// TIA Portal project "Tia-portal-PLC" (V16)

(* hardware
DEVICE "S71500/ET200MP station_1"  S7-1500 station
   slot 0: "Rail_0"  Rack  6ES7 590-1***0-0AA0
   slot 1: "PLC_1"  CPU 1512C-1 PN  6ES7 512-1CK01-0AB0  V2.8
      slot 3: "CPU display_1"  6ES7591-1AA00-0AA0
      slot 32768: "PROFINET interface_1"  X1
         slot 32769: "Port_1"  X1 P1
         slot 32770: "Port_2"  X1 P2
      slot 34817: "Virtual CP interface port_1"  Virtual CP interface port  Virtual CP interface port
DEVICE "S71500/ET200MP station_2"  S7-1500 station
   slot 0: "Rail_0"  Rack  6ES7 590-1***0-0AA0
   slot 1: "PLC_2"  CPU 1512C-1 PN  6ES7 512-1CK01-0AB0  V2.8
      slot 3: "CPU display_1"  6ES7591-1AA00-0AA0
      slot 32768: "PROFINET interface_1"  X1
         slot 32769: "Port_1"  X1 P1
         slot 32770: "Port_2"  X1 P2
      slot 34817: "Virtual CP interface port_1"  Virtual CP interface port  Virtual CP interface port
DEVICE "HMI_1"  TP700 Comfort
   slot 0: "HMI_1"  TP700 Comfort  6AV2 124-0GC01-0AX0  16.0.0.0
   slot 1: "HMI_RT_1"  TP700 Comfort  6AV2 124-0GC01-0AX0  16.0.0.0
   slot 5: "HMI_1.IE_CP_1"  PROFINET Interface  16.0.0.0
      slot 1: "PROFINET Interface_1"  PROFINET Interface
         slot 1: "Port_1"  Port
         slot 2: "Port_2"  Port
   slot 7: "HMI_1.MPI/DP_CP_1"  MPI/DP Interface  16.0.0.0
*)

// ===== PLC "PLC_1"  CPU 1512C-1 PN =====

VAR_GLOBAL   // PLC tag table "Default tag table"
   "Tag_1" AT %M0.0 : Bool;
END_VAR

VAR_GLOBAL   // PLC tag table "Inputs"
   "Start_pos" AT %I0.0 : Bool;   // Item in starting position
   "Size_measure_pos" AT %I0.1 : Bool;   // Item in size measuring position
   "Weight_mes_pos" AT %I0.2 : Bool;   // Item in weight measuring pisition
   "Servo_table_pos" AT %I0.3 : Bool;   // Item on servo controlled table
   "Metal_sensor" AT %I0.4 : Bool;   // Inductive sensor
   "Grip_cyl_end_ext" AT %I0.5 : Bool;   // Reed sensor. Gripping cylinder in end position is extended
   "Grip_cyl_end_ret" AT %I0.6 : Bool;   // Reed sensor. Gripping cylinder in end position is retracted
   "Cyl_at_table_ext" AT %I0.7 : Bool;   // Reed sensor. Cylinder, pushing in bin is extended
   "Cyl_at_table_ret" AT %I1.0 : Bool;   // Reed sensor. Cylinder, pushing in bin is retracted
   "ES1" AT %I1.7 : Bool;   // Emergency stop button for measuring
   "ES2" AT %I2.0 : Bool;   // Emergency stop button for sorting
   "Size_measure" AT %IW0 : Int;   // Size measuring sensor
   "Load_cell" AT %IW2 : Int;   // Load cell
   "Grip_cyl_start_ext" AT %I2.1 : Bool;   // Reed sensor. Gripping cylinder in starting position is extended
   "Grip_cyl_start_ret" AT %I2.2 : Bool;   // Reed sensor. Gripping cylinder in starting position is retracted
   "Control24VButton" AT %I2.3 : Bool;   // Giving 24V supply for output moduls
   "Metal_measure_pos" AT %I2.4 : Bool;   // Item in metal measuring position
   "End_pos_at_conveyor" AT %I2.5 : Bool;   // Item in end position at inverter controlled conveyor
END_VAR

VAR_GLOBAL   // PLC tag table "Outputs"
   "Green_light" AT %Q4.0 : Bool;   // Green light
   "Yellow_light" AT %Q4.1 : Bool;   // Yellow light
   "Red_light" AT %Q4.2 : Bool;   // Red light
   "Move_grip_cyl_end_fwd" AT %Q4.3 : Bool;   // Extend gripping cylinder in end position
   "Move_grip_cyl_end_bwd" AT %Q4.4 : Bool;   // Retract gripping cylinder in end position
   "Move_cyl_at_table_fwd" AT %Q4.5 : Bool;   // Extend cylinder 1 for bin
   "Move_cyl_at_table_bwd" AT %Q4.6 : Bool;   // Retract cylinder 1 for bin
   "Conveyor_forward" AT %Q5.5 : Bool;   // Output for the inverter. Move conveyor forward
   "Conveyor_backward" AT %Q5.6 : Bool;   // Output for the inverter. Move conveyor backward
   "Move_grip_cyl_start_fwd" AT %Q5.7 : Bool;   // Extend gripping cylinder in start position
   "Move_grip_cyl_start_bwd" AT %Q6.0 : Bool;   // Retract gripping cylinder in start position
   "Blue_light" AT %Q4.7 : Bool;
END_VAR

DATA_BLOCK "HMI-data"   // DB2
{ S7_Optimized_Access := 'TRUE' }
VERSION : 0.1
   VAR
      AutomaticMode : Bool;
      StartConveyor : Bool;
      StopConveyor : Bool;
      ItemInTheSystem : Bool;   // If there is an item in the system
      TableAtHome : Bool;
      TableAtBin1 : Bool;
      TableAtBin2 : Bool;
      TableAtBin3 : Bool;
      TableAtBin4 : Bool;
      ES1NC : Bool := true;   // Emergency button for simulation
      ES2NC : Bool := true;   // Emergency button for simulation
      ControlSupplyOK : Bool;   // Control 24V for simulation
      SizeInCm : Real;
      MetalMaterial : Bool;
      WeightInKg : Real;
      Bin1Breed : Bool;   // Small and non metal
      Bin2Breed : Bool;   // Small and metal
      Bin3Breed : Bool;   // Large and not metal
      Bin4Breed : Bool;   // Large and metal
      HomePosition : LReal;
      Bin1Position : LReal := 30.0;
      Bin2Position : LReal := 60.0;
      Bin3Postion : LReal := 90.0;
      Bin4Position : LReal := 120.0;
   END_VAR
BEGIN
END_DATA_BLOCK

DATA_BLOCK "OPCUA-data"   // DB4
{ S7_Optimized_Access := 'FALSE' }
VERSION : 0.1
   VAR
      Sensor1 : Bool := true;
   END_VAR
BEGIN
END_DATA_BLOCK

DATA_BLOCK "Sorting-motion-control_DB"   // DB7
{ S7_Optimized_Access := 'TRUE' }
VERSION : 0.1
// stored: InstanceOfName Sorting-motion-control
"Sorting-motion-control"
BEGIN
END_DATA_BLOCK

DATA_BLOCK "Size-measure_DB"   // DB8
{ S7_Optimized_Access := 'TRUE' }
VERSION : 0.1
// stored: InstanceOfName Size-measure
"Size-measure"
BEGIN
END_DATA_BLOCK

DATA_BLOCK "Weight-measure_DB"   // DB9
{ S7_Optimized_Access := 'TRUE' }
VERSION : 0.1
// stored: InstanceOfName Weight-measure
"Weight-measure"
BEGIN
END_DATA_BLOCK

DATA_BLOCK "Bin-sensors-from-PLC2"   // DB14
{ S7_Optimized_Access := 'FALSE' }
VERSION : 0.1
   VAR
      Bin1Full : Bool;
      Bin2Full : Bool;
      Bin3Full : Bool;
      Bin4Full : Bool;
   END_VAR
BEGIN
END_DATA_BLOCK

DATA_BLOCK "PLC2-communication_DB"   // DB16
{ S7_Optimized_Access := 'TRUE' }
VERSION : 0.1
// stored: InstanceOfName PLC2-communication
"PLC2-communication"
BEGIN
END_DATA_BLOCK

// folder: System blocks/Program resources

DATA_BLOCK "Start-pos-timer-DB"   // DB3
{ S7_Optimized_Access := 'TRUE' }
AUTHOR : Simatic
FAMILY : IEC
NAME : IEC_TMR
VERSION : 1.0
// stored: InstanceOfName IEC_TIMER
"IEC_TIMER"
BEGIN
END_DATA_BLOCK

DATA_BLOCK "IEC_Timer_0_DB"   // DB5
{ S7_Optimized_Access := 'TRUE' }
AUTHOR : Simatic
FAMILY : IEC
NAME : IEC_TMR
VERSION : 1.0
// stored: InstanceOfName IEC_TIMER
"IEC_TIMER"
BEGIN
END_DATA_BLOCK

DATA_BLOCK "IEC_Timer_0_DB_1"   // DB6
{ S7_Optimized_Access := 'TRUE' }
AUTHOR : Simatic
FAMILY : IEC
NAME : IEC_TMR
VERSION : 1.0
// stored: InstanceOfName IEC_TIMER
"IEC_TIMER"
BEGIN
END_DATA_BLOCK

DATA_BLOCK "IEC_Timer_0_DB_2"   // DB10
{ S7_Optimized_Access := 'TRUE' }
AUTHOR : Simatic
FAMILY : IEC
NAME : IEC_TMR
VERSION : 1.0
// stored: InstanceOfName IEC_TIMER
"IEC_TIMER"
BEGIN
END_DATA_BLOCK

DATA_BLOCK "IEC_Timer_0_DB_3"   // DB11
{ S7_Optimized_Access := 'TRUE' }
AUTHOR : Simatic
FAMILY : IEC
NAME : IEC_TMR
VERSION : 1.0
// stored: InstanceOfName IEC_TIMER
"IEC_TIMER"
BEGIN
END_DATA_BLOCK

DATA_BLOCK "IEC_Timer_0_DB_5"   // DB13
{ S7_Optimized_Access := 'TRUE' }
AUTHOR : Simatic
FAMILY : IEC
NAME : IEC_TMR
VERSION : 1.0
// stored: InstanceOfName IEC_TIMER
"IEC_TIMER"
BEGIN
END_DATA_BLOCK

DATA_BLOCK "PLC_1_Receive_DB"   // DB15
{ S7_Optimized_Access := 'TRUE' }
AUTHOR : SIMATIC
FAMILY : MC7Plus
NAME : TC_IP_v4
VERSION : 1.0
// stored: InstanceOfName TCON_IP_v4
"TCON_IP_v4"
BEGIN
   ID := 1;
   InterfaceId := 64;
   LocalPort := 2000;
   RemoteAddress.ADDR[1] := 192;
   RemoteAddress.ADDR[2] := 168;
   RemoteAddress.ADDR[4] := 14;
END_DATA_BLOCK

DATA_BLOCK "IEC_Timer_0_DB_8"   // DB17
{ S7_Optimized_Access := 'TRUE' }
AUTHOR : Simatic
FAMILY : IEC
NAME : IEC_TMR
VERSION : 1.0
// stored: InstanceOfName IEC_TIMER
"IEC_TIMER"
BEGIN
END_DATA_BLOCK

DATA_BLOCK "IEC_Timer_0_DB_6"   // DB18
{ S7_Optimized_Access := 'TRUE' }
AUTHOR : Simatic
FAMILY : IEC
NAME : IEC_TMR
VERSION : 1.0
// stored: InstanceOfName IEC_TIMER
"IEC_TIMER"
BEGIN
END_DATA_BLOCK

DATA_BLOCK "IEC_Timer_0_DB_7"   // DB19
{ S7_Optimized_Access := 'TRUE' }
AUTHOR : Simatic
FAMILY : IEC
NAME : IEC_TMR
VERSION : 1.0
// stored: InstanceOfName IEC_TIMER
"IEC_TIMER"
BEGIN
END_DATA_BLOCK

// folder: (top level)

DATA_BLOCK "SortingAxis_1"   // DB1, Motion_DB
{ S7_Optimized_Access := 'TRUE' }
AUTHOR : SIMATIC
FAMILY : MC_1500
VERSION : 5.0
// stored: InstanceOfName TO_PositioningAxis
"TO_PositioningAxis"
BEGIN
END_DATA_BLOCK

FUNCTION_BLOCK "Sorting-motion-control"   // FB1, LAD
{ S7_Optimized_Access := 'TRUE' }
VERSION : 0.1
   VAR_INPUT
      EnablePower : Bool;
      ExecuteReset : Bool;
      ExecuteHome : Bool;
      ExecuteHalt : Bool;
      JogFwd : Bool;
      JogBwd : Bool;
      JogVelocity : LReal;
      ExecuteMoveVelocity : Bool;
      McVelocity : LReal;
      ExecuteMoveRelative : Bool;
      MoveRelativeValue : LReal;
      ExecuteMoveAbsolute : Bool;
      MoveAbsoluteValue : LReal;
      ExecuteStop : Bool;
   END_VAR
   VAR_OUTPUT
      ActualPosition : LReal;
      ActualSpeed : LReal;
      ActualVelocity : LReal;
   END_VAR
   VAR
      MC_POWER_Instance : MC_POWER;
      MC_RESET_Instance : MC_RESET;
      MC_HOME_Instance : MC_HOME;
      MC_HALT_Instance : MC_HALT;
      MC_MOVEJOG_Instance : MC_MOVEJOG;
      MC_MOVEVELOCITY_Instance : MC_MOVEVELOCITY;
      MC_MOVERELATIVE_Instance : MC_MOVERELATIVE;
      MC_MOVEABSOLUTE_Instance : MC_MOVEABSOLUTE;
      MC_STOP_Instance : MC_STOP;
   END_VAR
BEGIN

REGION Network 1: MC Power
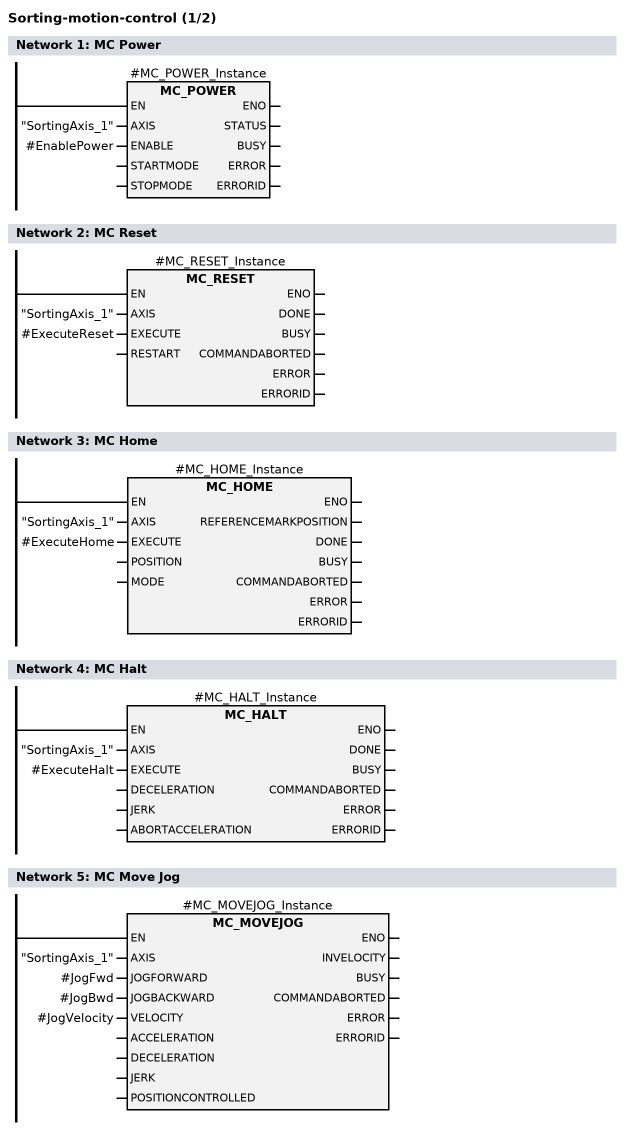
   #MC_POWER_Instance(Axis := "SortingAxis_1", Enable := #EnablePower);   // MC_POWER
END_REGION

REGION Network 2: MC Reset
   #MC_RESET_Instance(Axis := "SortingAxis_1", Execute := #ExecuteReset);   // MC_RESET
END_REGION

REGION Network 3: MC Home
   #MC_HOME_Instance(Axis := "SortingAxis_1", Execute := #ExecuteHome);   // MC_HOME
END_REGION

REGION Network 4: MC Halt
   #MC_HALT_Instance(Axis := "SortingAxis_1", Execute := #ExecuteHalt);   // MC_HALT
END_REGION

REGION Network 5: MC Move Jog
   #MC_MOVEJOG_Instance(Axis := "SortingAxis_1",   // MC_MOVEJOG
                        JogForward := #JogFwd,
                        JogBackward := #JogBwd,
                        Velocity := #JogVelocity);
END_REGION

REGION Network 6: MC Move Velocity
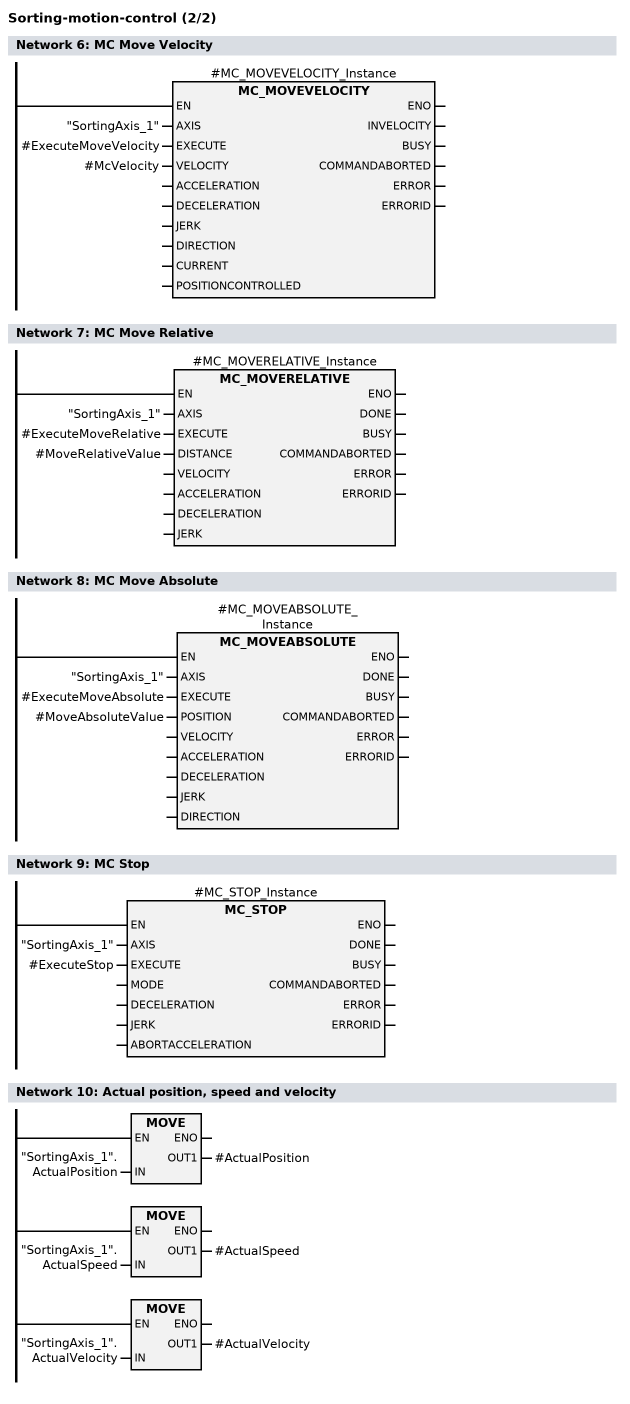
   #MC_MOVEVELOCITY_Instance(Axis := "SortingAxis_1", Execute := #ExecuteMoveVelocity, Velocity := #McVelocity);   // MC_MOVEVELOCITY
END_REGION

REGION Network 7: MC Move Relative
   #MC_MOVERELATIVE_Instance(Axis := "SortingAxis_1",   // MC_MOVERELATIVE
                           Execute := #ExecuteMoveRelative,
                           Distance := #MoveRelativeValue);
END_REGION

REGION Network 8: MC Move Absolute
   #MC_MOVEABSOLUTE_Instance(Axis := "SortingAxis_1",   // MC_MOVEABSOLUTE
                           Execute := #ExecuteMoveAbsolute,
                           Position := #MoveAbsoluteValue);
END_REGION

REGION Network 9: MC Stop
   #MC_STOP_Instance(Axis := "SortingAxis_1", Execute := #ExecuteStop);   // MC_STOP
END_REGION

REGION Network 10: Actual position, speed and velocity
   RUNG wire#powerrail
      Move(in := "SortingAxis_1".ActualPosition, out1 => #ActualPosition)
   END_RUNG
   RUNG wire#powerrail
      Move(in := "SortingAxis_1".ActualSpeed, out1 => #ActualSpeed)
   END_RUNG
   RUNG wire#powerrail
      Move(in := "SortingAxis_1".ActualVelocity, out1 => #ActualVelocity)
   END_RUNG
   // the same network as SCL:
   #ActualPosition := "SortingAxis_1".ActualPosition;
   #ActualSpeed := "SortingAxis_1".ActualSpeed;
   #ActualVelocity := "SortingAxis_1".ActualVelocity;
END_REGION
END_FUNCTION_BLOCK

FUNCTION_BLOCK "Size-measure"   // FB2, LAD
{ S7_Optimized_Access := 'TRUE' }
VERSION : 0.1
   VAR_INPUT
      TestValue : Int := 0;
   END_VAR
   VAR_OUTPUT
      SizeInCm : Real;
   END_VAR
   VAR_TEMP
      SizeInPercent : Real;
   END_VAR
BEGIN

REGION Network 1
   // Converting analog voltage to percent
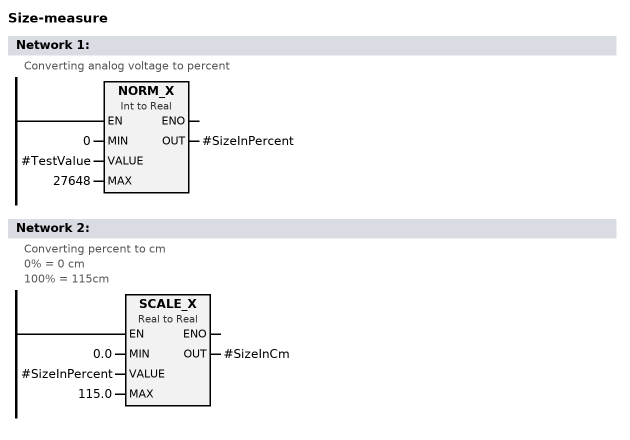
   RUNG wire#powerrail
      { S7_Templates := "[SrcType := Int, DestType := Real]" } Normalize(min := 0, value := #TestValue, max := 27648, out => #SizeInPercent)
   END_RUNG
   // the same network as SCL:
   #SizeInPercent := NORM_X(MIN := 0, VALUE := #TestValue, MAX := 27648);
END_REGION

REGION Network 2
   // Converting percent to cm
   // 0% = 0 cm
   // 100% = 115cm
   RUNG wire#powerrail
      { S7_Templates := "[SrcType := Real, DestType := Real]" } Scale(min := 0.0, value := #SizeInPercent, max := 115.0, out => #SizeInCm)
   END_RUNG
   // the same network as SCL:
   #SizeInCm := SCALE_X(MIN := 0.0, VALUE := #SizeInPercent, MAX := 115.0);
END_REGION
END_FUNCTION_BLOCK

FUNCTION_BLOCK "Weight-measure"   // FB3, LAD
{ S7_Optimized_Access := 'TRUE' }
VERSION : 0.1
   VAR_INPUT
      TestValue : Int := 0;
   END_VAR
   VAR_OUTPUT
      WeightInKg : Real;
   END_VAR
   VAR_TEMP
      WeightInPercent : Real;
   END_VAR
BEGIN

REGION Network 1
   // Converting analog voltage to percent
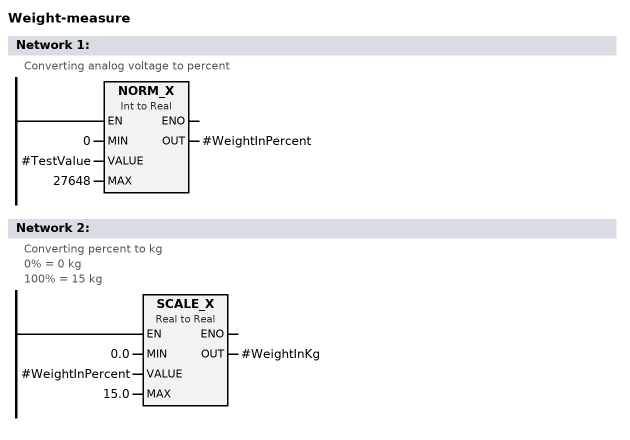
   RUNG wire#powerrail
      { S7_Templates := "[SrcType := Int, DestType := Real]" } Normalize(min := 0, value := #TestValue, max := 27648, out => #WeightInPercent)
   END_RUNG
   // the same network as SCL:
   #WeightInPercent := NORM_X(MIN := 0, VALUE := #TestValue, MAX := 27648);
END_REGION

REGION Network 2
   // Converting percent to kg
   // 0% = 0 kg
   // 100% = 15 kg
   RUNG wire#powerrail
      { S7_Templates := "[SrcType := Real, DestType := Real]" } Scale(min := 0.0, value := #WeightInPercent, max := 15.0, out => #WeightInKg)
   END_RUNG
   // the same network as SCL:
   #WeightInKg := SCALE_X(MIN := 0.0, VALUE := #WeightInPercent, MAX := 15.0);
END_REGION
END_FUNCTION_BLOCK

FUNCTION_BLOCK "PLC2-communication"   // FB4, LAD
TITLE = Communication with PLC2
{ S7_Optimized_Access := 'TRUE' }
VERSION : 0.1
   VAR_INPUT
      EnableConnAndRead : Bool;
   END_VAR
   VAR
      TRCV_C_Instance : TRCV_C;
   END_VAR
BEGIN

REGION Network 1
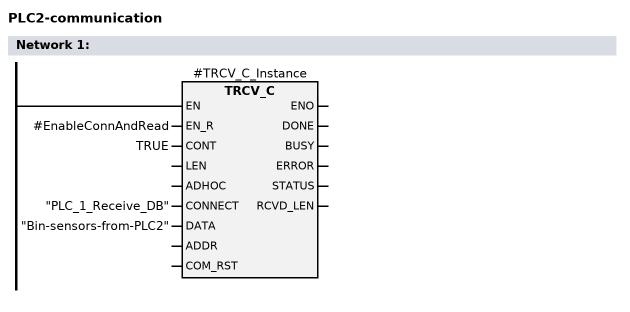
   #TRCV_C_Instance(EN_R := #EnableConnAndRead,   // TRCV_C
                    CONT := TRUE,
                    CONNECT := "PLC_1_Receive_DB",
                    DATA := "Bin-sensors-from-PLC2");
END_REGION
END_FUNCTION_BLOCK

FUNCTION "Home-positions" : Void   // FC1, LAD
{ S7_Optimized_Access := 'TRUE' }
VERSION : 0.1
// If there is 24V control power supply, everything goes to home position.
// If the ControlSupplyOK variable is true.
BEGIN

REGION Network 1: Extend gripping cylinder in start position
   // Gripping cylinder in start position is extended
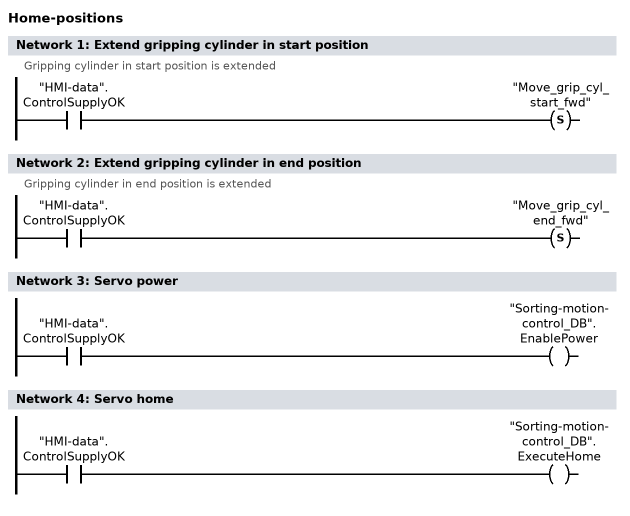
   RUNG wire#powerrail
      Contact( "HMI-data".ControlSupplyOK )
      S_Coil( "Move_grip_cyl_start_fwd" )
   END_RUNG
   // the same network as SCL:
   IF "HMI-data".ControlSupplyOK THEN "Move_grip_cyl_start_fwd" := TRUE; END_IF;
END_REGION

REGION Network 2: Extend gripping cylinder in end position
   // Gripping cylinder in end position is extended
   RUNG wire#powerrail
      Contact( "HMI-data".ControlSupplyOK )
      S_Coil( "Move_grip_cyl_end_fwd" )
   END_RUNG
   // the same network as SCL:
   IF "HMI-data".ControlSupplyOK THEN "Move_grip_cyl_end_fwd" := TRUE; END_IF;
END_REGION

REGION Network 3: Servo power
   RUNG wire#powerrail
      Contact( "HMI-data".ControlSupplyOK )
      Coil( "Sorting-motion-control_DB".EnablePower )
   END_RUNG
   // the same network as SCL:
   "Sorting-motion-control_DB".EnablePower := "HMI-data".ControlSupplyOK;
END_REGION

REGION Network 4: Servo home
   RUNG wire#powerrail
      Contact( "HMI-data".ControlSupplyOK )
      Coil( "Sorting-motion-control_DB".ExecuteHome )
   END_RUNG
   // the same network as SCL:
   "Sorting-motion-control_DB".ExecuteHome := "HMI-data".ControlSupplyOK;
END_REGION
END_FUNCTION

FUNCTION "Control24V" : Void   // FC2, LAD
{ S7_Optimized_Access := 'TRUE' }
VERSION : 0.1
BEGIN

REGION Network 1: Control 24V for simulation
   // This is the simulation of the safety circuit. Power supply for the output modules.
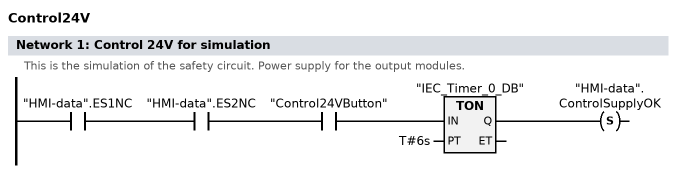
   "IEC_Timer_0_DB".TON(IN := "HMI-data".ES1NC AND "HMI-data".ES2NC AND "Control24VButton", PT := T#6s);
   IF "IEC_Timer_0_DB".Q THEN "HMI-data".ControlSupplyOK := TRUE; END_IF;
END_REGION
END_FUNCTION

FUNCTION "Table-positions" : Void   // FC3, LAD
{ S7_Optimized_Access := 'TRUE' }
VERSION : 0.1
BEGIN

REGION Network 1: Home position
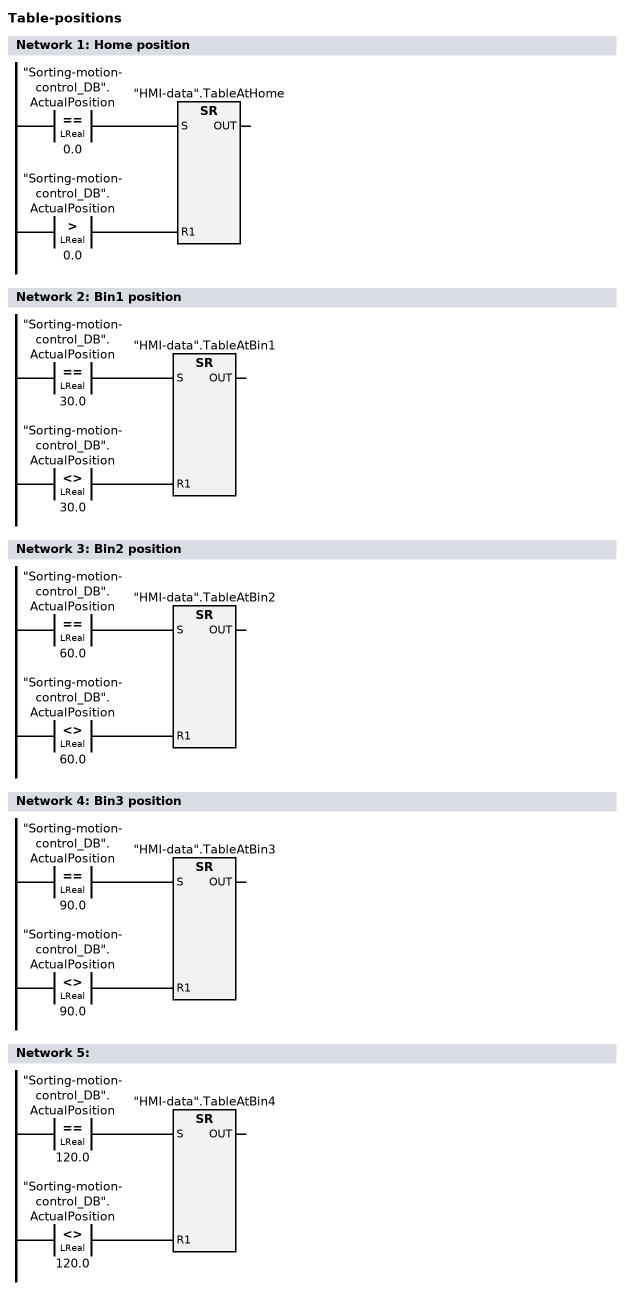
   RUNG wire#powerrail
      { S7_Templates := "SrcType := LReal" } EQ_Contact(in1 := "Sorting-motion-control_DB".ActualPosition, in2 := 0.0)
      S_SR(operand := "HMI-data".TableAtHome, r1 := wire#w1)
   END_RUNG
   RUNG wire#powerrail
      { S7_Templates := "SrcType := LReal" } GT_Contact(in1 := "Sorting-motion-control_DB".ActualPosition, in2 := 0.0)
   END_RUNG wire#w1
   // the same network as SCL:
   IF "Sorting-motion-control_DB".ActualPosition = 0.0 THEN
       "HMI-data".TableAtHome := TRUE;   // SR flip-flop
   END_IF;
   IF "Sorting-motion-control_DB".ActualPosition > 0.0 THEN "HMI-data".TableAtHome := FALSE; END_IF;
END_REGION

REGION Network 2: Bin1 position
   RUNG wire#powerrail
      { S7_Templates := "SrcType := LReal" } EQ_Contact(in1 := "Sorting-motion-control_DB".ActualPosition, in2 := 30.0)
      S_SR(operand := "HMI-data".TableAtBin1, r1 := wire#w1)
   END_RUNG
   RUNG wire#powerrail
      { S7_Templates := "SrcType := LReal" } NE_Contact(in1 := "Sorting-motion-control_DB".ActualPosition, in2 := 30.0)
   END_RUNG wire#w1
   // the same network as SCL:
   IF "Sorting-motion-control_DB".ActualPosition = 30.0 THEN
       "HMI-data".TableAtBin1 := TRUE;   // SR flip-flop
   END_IF;
   IF "Sorting-motion-control_DB".ActualPosition <> 30.0 THEN "HMI-data".TableAtBin1 := FALSE; END_IF;
END_REGION

REGION Network 3: Bin2 position
   RUNG wire#powerrail
      { S7_Templates := "SrcType := LReal" } EQ_Contact(in1 := "Sorting-motion-control_DB".ActualPosition, in2 := 60.0)
      S_SR(operand := "HMI-data".TableAtBin2, r1 := wire#w1)
   END_RUNG
   RUNG wire#powerrail
      { S7_Templates := "SrcType := LReal" } NE_Contact(in1 := "Sorting-motion-control_DB".ActualPosition, in2 := 60.0)
   END_RUNG wire#w1
   // the same network as SCL:
   IF "Sorting-motion-control_DB".ActualPosition = 60.0 THEN
       "HMI-data".TableAtBin2 := TRUE;   // SR flip-flop
   END_IF;
   IF "Sorting-motion-control_DB".ActualPosition <> 60.0 THEN "HMI-data".TableAtBin2 := FALSE; END_IF;
END_REGION

REGION Network 4: Bin3 position
   RUNG wire#powerrail
      { S7_Templates := "SrcType := LReal" } EQ_Contact(in1 := "Sorting-motion-control_DB".ActualPosition, in2 := 90.0)
      S_SR(operand := "HMI-data".TableAtBin3, r1 := wire#w1)
   END_RUNG
   RUNG wire#powerrail
      { S7_Templates := "SrcType := LReal" } NE_Contact(in1 := "Sorting-motion-control_DB".ActualPosition, in2 := 90.0)
   END_RUNG wire#w1
   // the same network as SCL:
   IF "Sorting-motion-control_DB".ActualPosition = 90.0 THEN
       "HMI-data".TableAtBin3 := TRUE;   // SR flip-flop
   END_IF;
   IF "Sorting-motion-control_DB".ActualPosition <> 90.0 THEN "HMI-data".TableAtBin3 := FALSE; END_IF;
END_REGION

REGION Network 5
   RUNG wire#powerrail
      { S7_Templates := "SrcType := LReal" } EQ_Contact(in1 := "Sorting-motion-control_DB".ActualPosition, in2 := 120.0)
      S_SR(operand := "HMI-data".TableAtBin4, r1 := wire#w1)
   END_RUNG
   RUNG wire#powerrail
      { S7_Templates := "SrcType := LReal" } NE_Contact(in1 := "Sorting-motion-control_DB".ActualPosition, in2 := 120.0)
   END_RUNG wire#w1
   // the same network as SCL:
   IF "Sorting-motion-control_DB".ActualPosition = 120.0 THEN
       "HMI-data".TableAtBin4 := TRUE;   // SR flip-flop
   END_IF;
   IF "Sorting-motion-control_DB".ActualPosition <> 120.0 THEN "HMI-data".TableAtBin4 := FALSE; END_IF;
END_REGION
END_FUNCTION

FUNCTION "Breed-calculation" : Void   // FC4, LAD
{ S7_Optimized_Access := 'TRUE' }
VERSION : 0.1
BEGIN

REGION Network 1: Small and non metal
   // Bin1 breed
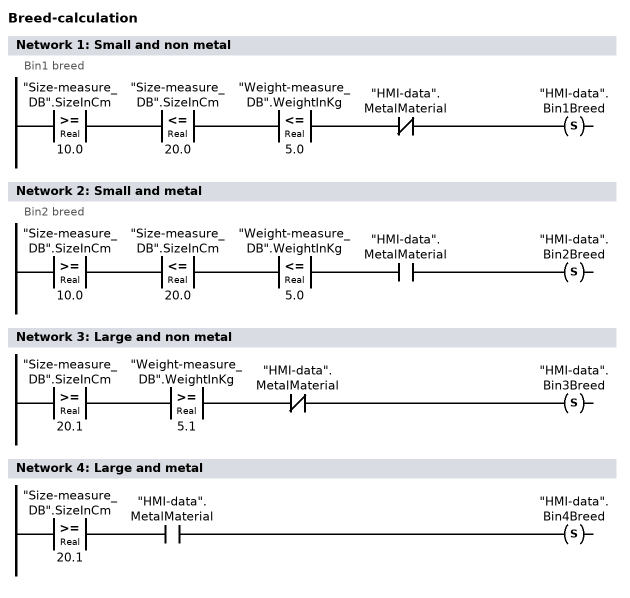
   RUNG wire#powerrail
      { S7_Templates := "SrcType := Real" } GE_Contact(in1 := "Size-measure_DB".SizeInCm, in2 := 10.0)
      { S7_Templates := "SrcType := Real" } LE_Contact(in1 := "Size-measure_DB".SizeInCm, in2 := 20.0)
      { S7_Templates := "SrcType := Real" } LE_Contact(in1 := "Weight-measure_DB".WeightInKg, in2 := 5.0)
      I_Contact( "HMI-data".MetalMaterial )
      S_Coil( "HMI-data".Bin1Breed )
   END_RUNG
   // the same network as SCL:
   IF ("Size-measure_DB".SizeInCm >= 10.0) AND ("Size-measure_DB".SizeInCm <= 20.0) AND ("Weight-measure_DB".WeightInKg <= 5.0) AND NOT "HMI-data".MetalMaterial THEN
       "HMI-data".Bin1Breed := TRUE;
   END_IF;
END_REGION

REGION Network 2: Small and metal
   // Bin2 breed
   RUNG wire#powerrail
      { S7_Templates := "SrcType := Real" } GE_Contact(in1 := "Size-measure_DB".SizeInCm, in2 := 10.0)
      { S7_Templates := "SrcType := Real" } LE_Contact(in1 := "Size-measure_DB".SizeInCm, in2 := 20.0)
      { S7_Templates := "SrcType := Real" } LE_Contact(in1 := "Weight-measure_DB".WeightInKg, in2 := 5.0)
      Contact( "HMI-data".MetalMaterial )
      S_Coil( "HMI-data".Bin2Breed )
   END_RUNG
   // the same network as SCL:
   IF ("Size-measure_DB".SizeInCm >= 10.0) AND ("Size-measure_DB".SizeInCm <= 20.0) AND ("Weight-measure_DB".WeightInKg <= 5.0) AND "HMI-data".MetalMaterial THEN
       "HMI-data".Bin2Breed := TRUE;
   END_IF;
END_REGION

REGION Network 3: Large and non metal
   RUNG wire#powerrail
      { S7_Templates := "SrcType := Real" } GE_Contact(in1 := "Size-measure_DB".SizeInCm, in2 := 20.1)
      { S7_Templates := "SrcType := Real" } GE_Contact(in1 := "Weight-measure_DB".WeightInKg, in2 := 5.1)
      I_Contact( "HMI-data".MetalMaterial )
      S_Coil( "HMI-data".Bin3Breed )
   END_RUNG
   // the same network as SCL:
   IF ("Size-measure_DB".SizeInCm >= 20.1) AND ("Weight-measure_DB".WeightInKg >= 5.1) AND NOT "HMI-data".MetalMaterial THEN
       "HMI-data".Bin3Breed := TRUE;
   END_IF;
END_REGION

REGION Network 4: Large and metal
   RUNG wire#powerrail
      { S7_Templates := "SrcType := Real" } GE_Contact(in1 := "Size-measure_DB".SizeInCm, in2 := 20.1)
      Contact( "HMI-data".MetalMaterial )
      S_Coil( "HMI-data".Bin4Breed )
   END_RUNG
   // the same network as SCL:
   IF ("Size-measure_DB".SizeInCm >= 20.1) AND "HMI-data".MetalMaterial THEN
       "HMI-data".Bin4Breed := TRUE;
   END_IF;
END_REGION
END_FUNCTION

ORGANIZATION_BLOCK "Main"   // OB1, LAD, ProgramCycle
TITLE = "Main Program Sweep (Cycle)"
{ S7_Optimized_Access := 'TRUE' }
VERSION : 0.1
   VAR_INPUT
      Initial_Call : Bool;   // Initial call of this OB
      Remanence : Bool;   // =True, if remanent data are available
   END_VAR
   VAR_TEMP   // added for the SCL form of the ladder/FBD networks
      _w1 : Bool;
      _w2 : Bool;
      _w3 : Bool;
      _w4 : Bool;
   END_VAR
BEGIN

REGION Network 1: Control 24V power supply
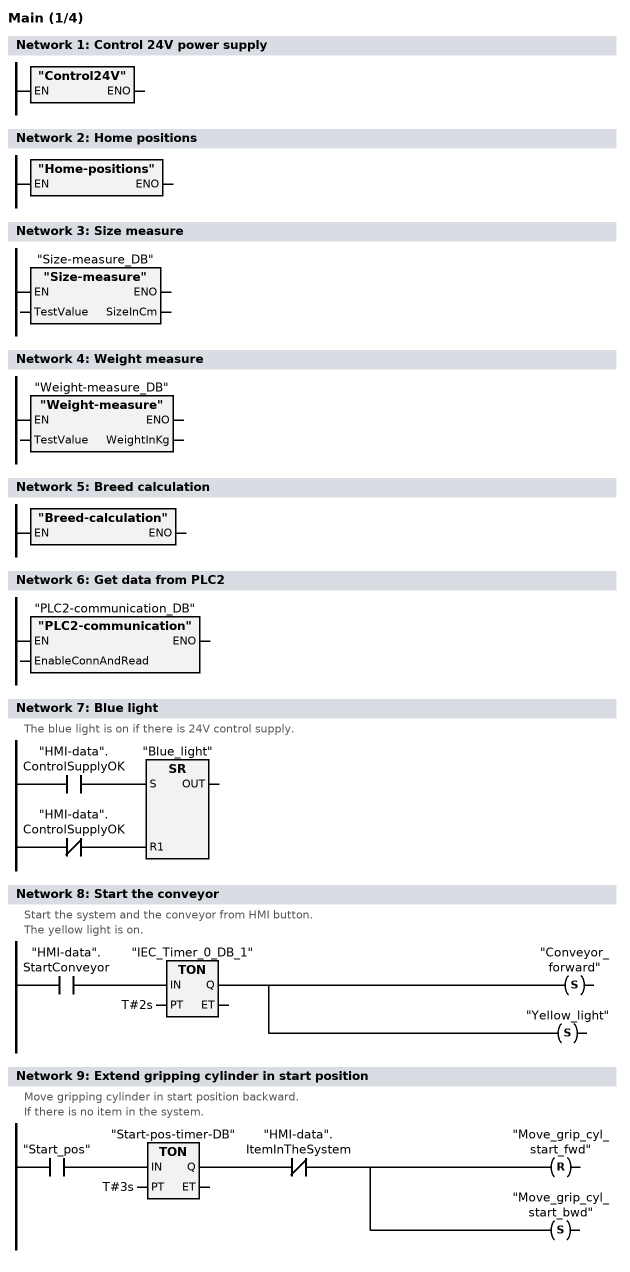
   RUNG wire#powerrail
      "Control24V"()
   END_RUNG
   // the same network as SCL:
   "Control24V"();
END_REGION

REGION Network 2: Home positions
   RUNG wire#powerrail
      "Home-positions"()
   END_RUNG
   // the same network as SCL:
   "Home-positions"();
END_REGION

REGION Network 3: Size measure
   RUNG wire#powerrail
      "Size-measure_DB"(TestValue :=, SizeInCm =>)
   END_RUNG
   // the same network as SCL:
   "Size-measure_DB"();   // "Size-measure"
END_REGION

REGION Network 4: Weight measure
   RUNG wire#powerrail
      "Weight-measure_DB"(TestValue :=, WeightInKg =>)
   END_RUNG
   // the same network as SCL:
   "Weight-measure_DB"();   // "Weight-measure"
END_REGION

REGION Network 5: Breed calculation
   RUNG wire#powerrail
      "Breed-calculation"()
   END_RUNG
   // the same network as SCL:
   "Breed-calculation"();
END_REGION

REGION Network 6: Get data from PLC2
   RUNG wire#powerrail
      "PLC2-communication_DB"(EnableConnAndRead :=)
   END_RUNG
   // the same network as SCL:
   "PLC2-communication_DB"();   // "PLC2-communication"
END_REGION

REGION Network 7: Blue light
   // The blue light is on if there is 24V control supply.
   RUNG wire#powerrail
      Contact( "HMI-data".ControlSupplyOK )
      S_SR(operand := "Blue_light", r1 := wire#w1)
   END_RUNG
   RUNG wire#powerrail
      I_Contact( "HMI-data".ControlSupplyOK )
   END_RUNG wire#w1
   // the same network as SCL:
   IF "HMI-data".ControlSupplyOK THEN
       "Blue_light" := TRUE;   // SR flip-flop
   END_IF;
   IF NOT "HMI-data".ControlSupplyOK THEN "Blue_light" := FALSE; END_IF;
END_REGION

REGION Network 8: Start the conveyor
   // Start the system and the conveyor from HMI button.
   // The yellow light is on.
   "IEC_Timer_0_DB_1".TON(IN := "HMI-data".StartConveyor, PT := T#2s);
   IF "IEC_Timer_0_DB_1".Q THEN
       "Conveyor_forward" := TRUE;
       "Yellow_light" := TRUE;
   END_IF;
END_REGION

REGION Network 9: Extend gripping cylinder in start position
   // Move gripping cylinder in start position backward.
   // If there is no item in the system.
   "Start-pos-timer-DB".TON(IN := "Start_pos", PT := T#3s);
   IF "Start-pos-timer-DB".Q AND NOT "HMI-data".ItemInTheSystem THEN
       "Move_grip_cyl_start_fwd" := FALSE;
       "Move_grip_cyl_start_bwd" := TRUE;
   END_IF;
END_REGION

REGION Network 10: If there is an item in the system
   // After leaving the start position sensor, the system is in progress so there is an item in the system.
   // The green light is on.
   // The yellow light is off.
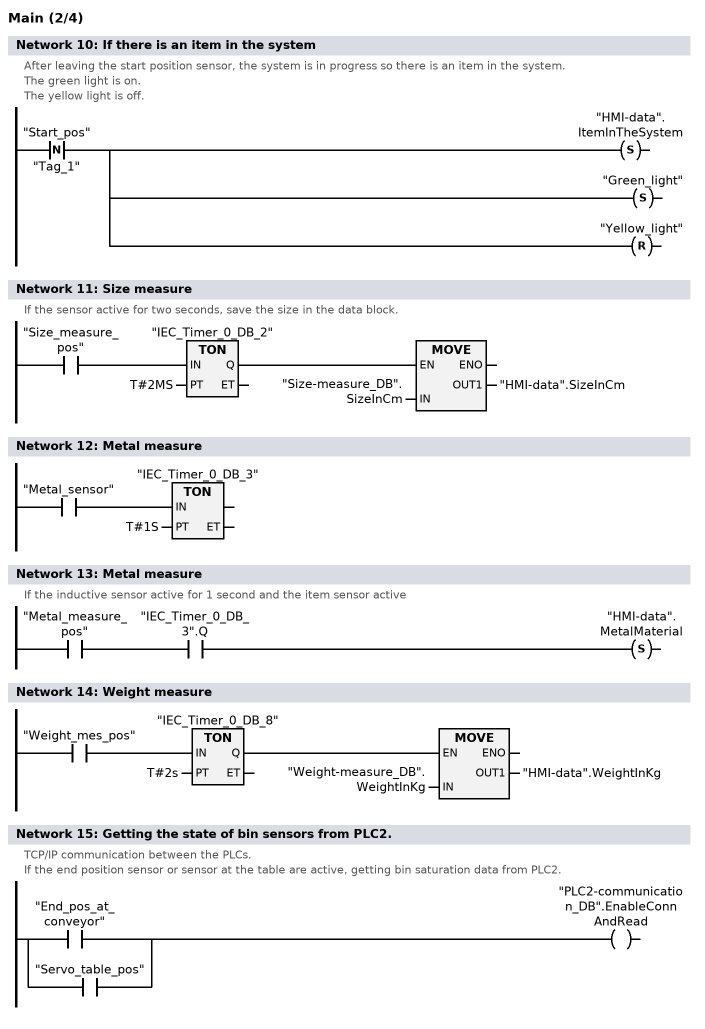
   RUNG wire#powerrail
      N_Contact(operand := "Start_pos", bit := "Tag_1")
      wire#w1
      S_Coil( "HMI-data".ItemInTheSystem )
   END_RUNG
   RUNG wire#w1
      S_Coil( "Green_light" )
   END_RUNG
   RUNG wire#w1
      R_Coil( "Yellow_light" )
   END_RUNG
   // the same network as SCL:
   #_w1 := NOT "Start_pos" AND "Tag_1";   // falling edge of "Start_pos"
   "Tag_1" := "Start_pos";
   IF #_w1 THEN
       "HMI-data".ItemInTheSystem := TRUE;
       "Green_light" := TRUE;
       "Yellow_light" := FALSE;
   END_IF;
END_REGION

REGION Network 11: Size measure
   // If the sensor active for two seconds, save the size in the data block.
   "IEC_Timer_0_DB_2".TON(IN := "Size_measure_pos", PT := T#2MS);
   IF "IEC_Timer_0_DB_2".Q THEN "HMI-data".SizeInCm := "Size-measure_DB".SizeInCm; END_IF;
END_REGION

REGION Network 12: Metal measure
   "IEC_Timer_0_DB_3".TON(IN := "Metal_sensor", PT := T#1S);
END_REGION

REGION Network 13: Metal measure
   // If the inductive sensor active for 1 second and the item sensor active
   RUNG wire#powerrail
      Contact( "Metal_measure_pos" )
      Contact( "IEC_Timer_0_DB_3".Q )
      S_Coil( "HMI-data".MetalMaterial )
   END_RUNG
   // the same network as SCL:
   IF "Metal_measure_pos" AND "IEC_Timer_0_DB_3".Q THEN "HMI-data".MetalMaterial := TRUE; END_IF;
END_REGION

REGION Network 14: Weight measure
   "IEC_Timer_0_DB_8".TON(IN := "Weight_mes_pos", PT := T#2s);
   IF "IEC_Timer_0_DB_8".Q THEN "HMI-data".WeightInKg := "Weight-measure_DB".WeightInKg; END_IF;
END_REGION

REGION Network 15: Getting the state of bin sensors from PLC2.
   // TCP/IP communication between the PLCs.
   // If the end position sensor or sensor at the table are active, getting bin saturation data from PLC2.
   RUNG wire#powerrail
      Contact( "End_pos_at_conveyor" )
      wire#w1
      Coil( "PLC2-communication_DB".EnableConnAndRead )
   END_RUNG
   RUNG wire#powerrail
      Contact( "Servo_table_pos" )
   END_RUNG wire#w1
   // the same network as SCL:
   "PLC2-communication_DB".EnableConnAndRead := "End_pos_at_conveyor" OR "Servo_table_pos";
END_REGION

REGION Network 16: Retract gripping cylinder in end position
   // If the sensor at conveyor is active for 1.5 seconds and the reed sensor is active and the certain bin is not full and the table is at home position.
   // The state of bin sensors comes from PLC2.
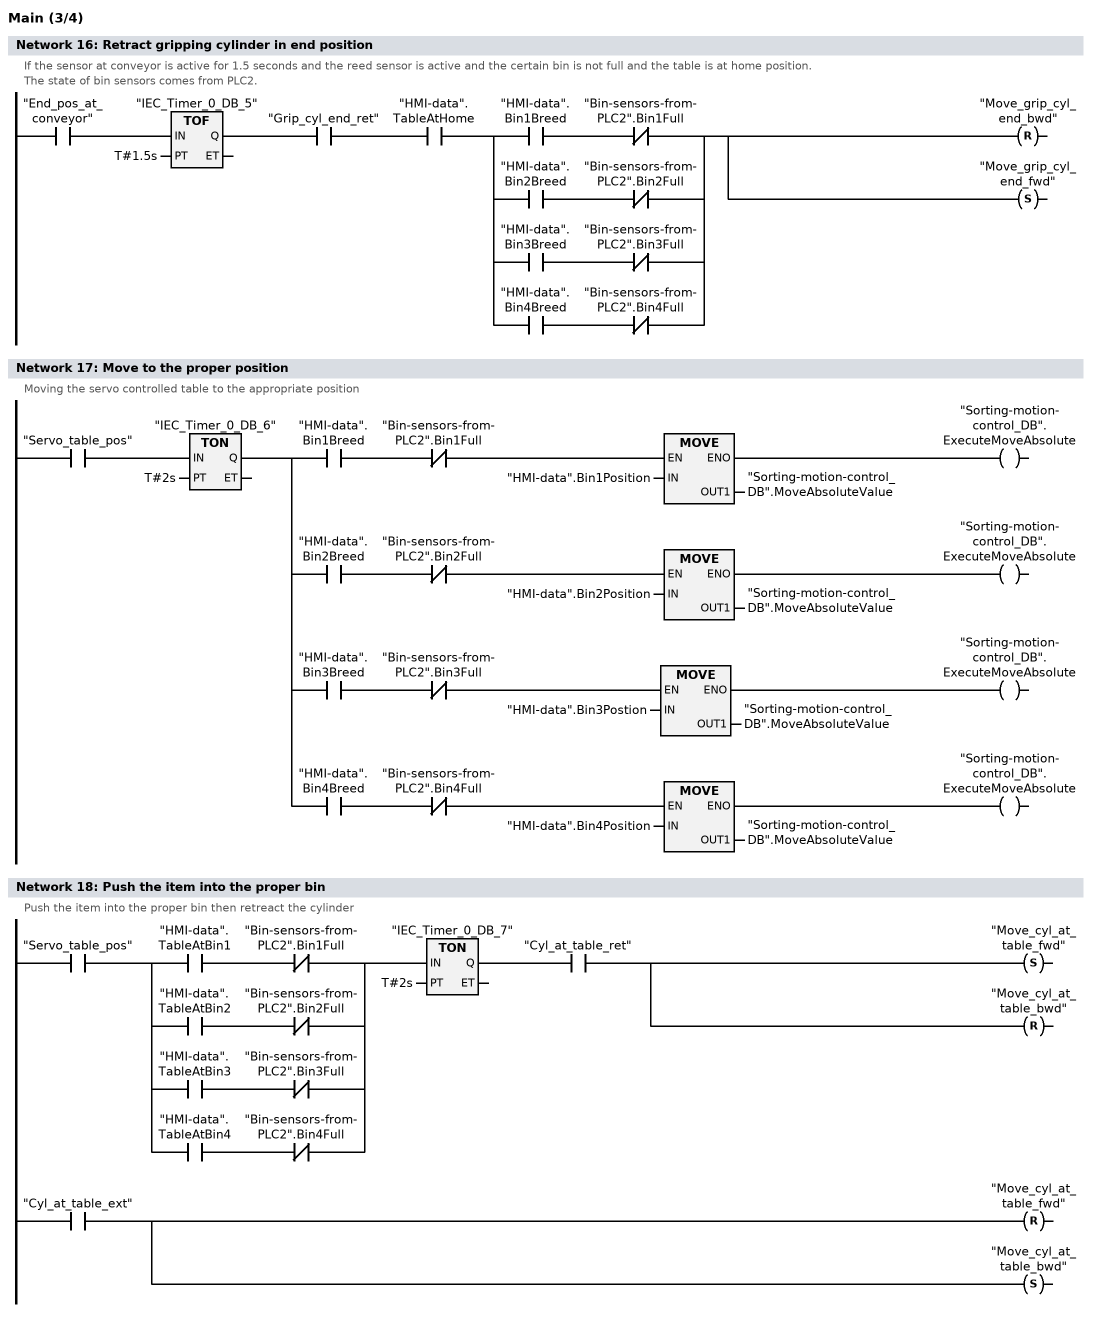
   "IEC_Timer_0_DB_5".TOF(IN := "End_pos_at_conveyor", PT := T#1.5s);
   IF "IEC_Timer_0_DB_5".Q AND "Grip_cyl_end_ret" AND "HMI-data".TableAtHome AND (("HMI-data".Bin1Breed AND NOT "Bin-sensors-from-PLC2".Bin1Full) OR ("HMI-data".Bin2Breed AND NOT "Bin-sensors-from-PLC2".Bin2Full) OR ("HMI-data".Bin3Breed AND NOT "Bin-sensors-from-PLC2".Bin3Full) OR ("HMI-data".Bin4Breed AND NOT "Bin-sensors-from-PLC2".Bin4Full)) THEN
       "Move_grip_cyl_end_bwd" := FALSE;
       "Move_grip_cyl_end_fwd" := TRUE;
   END_IF;
END_REGION

REGION Network 17: Move to the proper position
   // Moving the servo controlled table to the appropriate position
   "IEC_Timer_0_DB_6".TON(IN := "Servo_table_pos", PT := T#2s);
   #_w1 := "IEC_Timer_0_DB_6".Q AND "HMI-data".Bin1Breed AND NOT "Bin-sensors-from-PLC2".Bin1Full;
   IF #_w1 THEN "Sorting-motion-control_DB".MoveAbsoluteValue := "HMI-data".Bin1Position; END_IF;
   "Sorting-motion-control_DB".ExecuteMoveAbsolute := #_w1;
   #_w2 := "IEC_Timer_0_DB_6".Q AND "HMI-data".Bin2Breed AND NOT "Bin-sensors-from-PLC2".Bin2Full;
   IF #_w2 THEN "Sorting-motion-control_DB".MoveAbsoluteValue := "HMI-data".Bin2Position; END_IF;
   "Sorting-motion-control_DB".ExecuteMoveAbsolute := #_w2;
   #_w3 := "IEC_Timer_0_DB_6".Q AND "HMI-data".Bin3Breed AND NOT "Bin-sensors-from-PLC2".Bin3Full;
   IF #_w3 THEN "Sorting-motion-control_DB".MoveAbsoluteValue := "HMI-data".Bin3Postion; END_IF;
   "Sorting-motion-control_DB".ExecuteMoveAbsolute := #_w3;
   #_w4 := "IEC_Timer_0_DB_6".Q AND "HMI-data".Bin4Breed AND NOT "Bin-sensors-from-PLC2".Bin4Full;
   IF #_w4 THEN "Sorting-motion-control_DB".MoveAbsoluteValue := "HMI-data".Bin4Position; END_IF;
   "Sorting-motion-control_DB".ExecuteMoveAbsolute := #_w4;
END_REGION

REGION Network 18: Push the item into the proper bin
   // Push the item into the proper bin then retreact the cylinder
   "IEC_Timer_0_DB_7".TON(IN := "Servo_table_pos" AND (("HMI-data".TableAtBin1 AND NOT "Bin-sensors-from-PLC2".Bin1Full) OR ("HMI-data".TableAtBin2 AND NOT "Bin-sensors-from-PLC2".Bin2Full) OR ("HMI-data".TableAtBin3 AND NOT "Bin-sensors-from-PLC2".Bin3Full) OR ("HMI-data".TableAtBin4 AND NOT "Bin-sensors-from-PLC2".Bin4Full)),
                          PT := T#2s);
   IF "IEC_Timer_0_DB_7".Q AND "Cyl_at_table_ret" THEN
       "Move_cyl_at_table_fwd" := TRUE;
       "Move_cyl_at_table_bwd" := FALSE;
   END_IF;
   IF "Cyl_at_table_ext" THEN
       "Move_cyl_at_table_fwd" := FALSE;
       "Move_cyl_at_table_bwd" := TRUE;
   END_IF;
END_REGION

REGION Network 19: There is no item in the system any more.
   // The next item can move forward from the beginning of the conveyor.
   // The green light goes off.
   // The yellow light goes on.
   // Reset the parameters of the item.
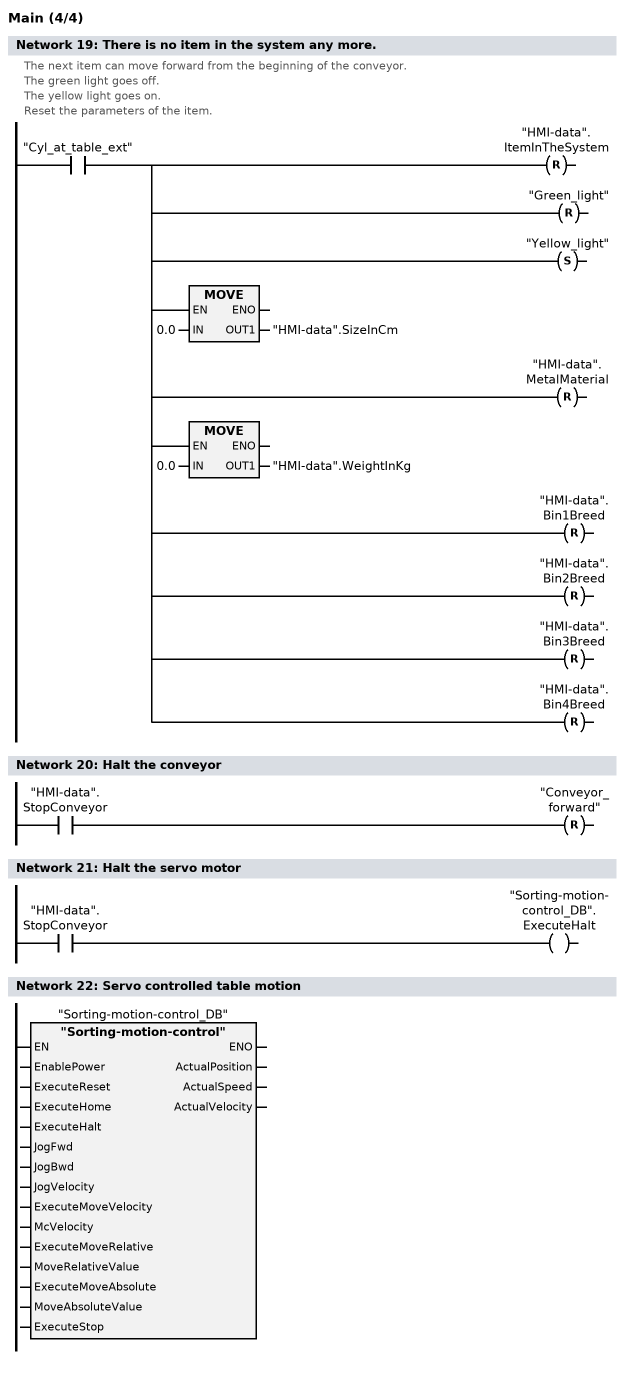
   RUNG wire#powerrail
      Contact( "Cyl_at_table_ext" )
      wire#w1
      R_Coil( "HMI-data".ItemInTheSystem )
   END_RUNG
   RUNG wire#w1
      R_Coil( "Green_light" )
   END_RUNG
   RUNG wire#w1
      S_Coil( "Yellow_light" )
   END_RUNG
   RUNG wire#w1
      Move(in := 0.0, out1 => "HMI-data".SizeInCm)
   END_RUNG
   RUNG wire#w1
      R_Coil( "HMI-data".MetalMaterial )
   END_RUNG
   RUNG wire#w1
      Move(in := 0.0, out1 => "HMI-data".WeightInKg)
   END_RUNG
   RUNG wire#w1
      R_Coil( "HMI-data".Bin1Breed )
   END_RUNG
   RUNG wire#w1
      R_Coil( "HMI-data".Bin2Breed )
   END_RUNG
   RUNG wire#w1
      R_Coil( "HMI-data".Bin3Breed )
   END_RUNG
   RUNG wire#w1
      R_Coil( "HMI-data".Bin4Breed )
   END_RUNG
   // the same network as SCL:
   IF "Cyl_at_table_ext" THEN
       "HMI-data".ItemInTheSystem := FALSE;
       "Green_light" := FALSE;
       "Yellow_light" := TRUE;
       "HMI-data".SizeInCm := 0.0;
       "HMI-data".MetalMaterial := FALSE;
       "HMI-data".WeightInKg := 0.0;
       "HMI-data".Bin1Breed := FALSE;
       "HMI-data".Bin2Breed := FALSE;
       "HMI-data".Bin3Breed := FALSE;
       "HMI-data".Bin4Breed := FALSE;
   END_IF;
END_REGION

REGION Network 20: Halt the conveyor
   RUNG wire#powerrail
      Contact( "HMI-data".StopConveyor )
      R_Coil( "Conveyor_forward" )
   END_RUNG
   // the same network as SCL:
   IF "HMI-data".StopConveyor THEN "Conveyor_forward" := FALSE; END_IF;
END_REGION

REGION Network 21: Halt the servo motor
   RUNG wire#powerrail
      Contact( "HMI-data".StopConveyor )
      Coil( "Sorting-motion-control_DB".ExecuteHalt )
   END_RUNG
   // the same network as SCL:
   "Sorting-motion-control_DB".ExecuteHalt := "HMI-data".StopConveyor;
END_REGION

REGION Network 22: Servo controlled table motion
   RUNG wire#powerrail
      "Sorting-motion-control_DB"(EnablePower :=, ExecuteReset :=, ExecuteHome :=, ExecuteHalt :=, JogFwd :=, JogBwd :=, JogVelocity :=, ExecuteMoveVelocity :=, McVelocity :=, ExecuteMoveRelative :=, MoveRelativeValue :=, ExecuteMoveAbsolute :=, MoveAbsoluteValue :=, ExecuteStop :=, ActualPosition =>, ActualSpeed =>, ActualVelocity =>)
   END_RUNG
   // the same network as SCL:
   "Sorting-motion-control_DB"();   // "Sorting-motion-control"
END_REGION
END_ORGANIZATION_BLOCK

// ===== PLC "PLC_2"  CPU 1512C-1 PN =====

DATA_BLOCK "Bin-sensors"   // DB1
{ S7_Optimized_Access := 'FALSE' }
VERSION : 0.1
   VAR
      Bin1Full : Bool;
      Bin2Full : Bool;
      Bin3Full : Bool;
      Bin4Full : Bool;
   END_VAR
BEGIN
END_DATA_BLOCK

// folder: System blocks/Program resources

DATA_BLOCK "PLC_2_Send_DB"   // DB2
{ S7_Optimized_Access := 'TRUE' }
AUTHOR : SIMATIC
FAMILY : MC7Plus
NAME : TC_IP_v4
VERSION : 1.0
// stored: InstanceOfName TCON_IP_v4
"TCON_IP_v4"
BEGIN
   ID := 1;
   InterfaceId := 64;
   RemotePort := 2000;
   ActiveEstablished := true;
   RemoteAddress.ADDR[1] := 192;
   RemoteAddress.ADDR[2] := 168;
   RemoteAddress.ADDR[4] := 11;
END_DATA_BLOCK

// folder: (top level)

FUNCTION_BLOCK "PLC1-communication"   // FB1, LAD
{ S7_Optimized_Access := 'TRUE' }
VERSION : 0.1
   VAR
      TSEND_C_Instance : TSEND_C;
   END_VAR
BEGIN

REGION Network 1
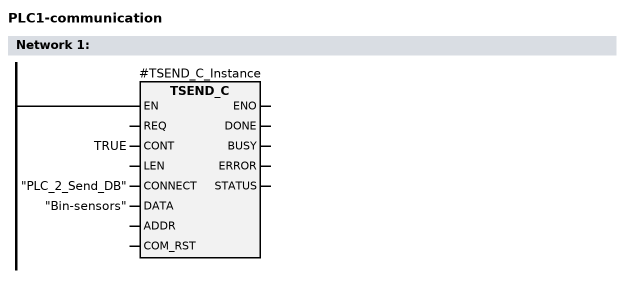
   #TSEND_C_Instance(CONT := TRUE, CONNECT := "PLC_2_Send_DB", DATA := "Bin-sensors");   // TSEND_C
END_REGION
END_FUNCTION_BLOCK

ORGANIZATION_BLOCK "Main"   // OB1, LAD, ProgramCycle
TITLE = "Main Program Sweep (Cycle)"
{ S7_Optimized_Access := 'TRUE' }
VERSION : 0.1
   VAR_INPUT
      Initial_Call : Bool;   // Initial call of this OB
      Remanence : Bool;   // =True, if remanent data are available
   END_VAR
BEGIN
END_ORGANIZATION_BLOCK

(* ===== HMI "HMI_RT_1" =====
system functions are stored by id; their names below are inferred from use
connection "HMI_Connection_1": ETHERNET, S7_1500_OMS
connection "HMI_Connection_2": ETHERNET, S7_1500_OMS

HMI tags "Default tag table"
   "Tag_ScreenNumber" : UInt, internal
   "Move_grip_cyl_start_fwd" : Bool = PLC Move_grip_cyl_start_fwd AT %Q5.7, 1 s

HMI tags "HMI-data"
   "HMI-data_AutomaticMode" : Bool = PLC "HMI-data".AutomaticMode, 1 s
   "HMI-data_StartConveyor" : Bool = PLC "HMI-data".StartConveyor, 1 s
   "HMI-data_StopConveyor" : Bool = PLC "HMI-data".StopConveyor, 1 s
   "HMI-data_SizeInCm" : Real = PLC "HMI-data".SizeInCm, 1 s
   "HMI-data_MetalMaterial" : Bool = PLC "HMI-data".MetalMaterial, 1 s
   "HMI-data_WeightInKg" : Real = PLC "HMI-data".WeightInKg, 1 s
   "HMI-data_TableAtHome" : Bool = PLC "HMI-data".TableAtHome, 1 s
   "HMI-data_TableAtBin1" : Bool = PLC "HMI-data".TableAtBin1, 1 s
   "HMI-data_TableAtBin2" : Bool = PLC "HMI-data".TableAtBin2, 1 s
   "HMI-data_TableAtBin3" : Bool = PLC "HMI-data".TableAtBin3, 1 s
   "HMI-data_TableAtBin4" : Bool = PLC "HMI-data".TableAtBin4, 1 s
   "HMI-data_ControlSupplyOK" : Bool = PLC "HMI-data".ControlSupplyOK, 1 s
   "HMI-data_ItemInTheSystem" : Bool = PLC "HMI-data".ItemInTheSystem, 1 s
   "HMI-data_Bin1Breed" : Bool = PLC "HMI-data".Bin1Breed, 1 s
   "HMI-data_Bin2Breed" : Bool = PLC "HMI-data".Bin2Breed, 1 s
   "HMI-data_Bin3Breed" : Bool = PLC "HMI-data".Bin3Breed, 1 s
   "HMI-data_Bin4Breed" : Bool = PLC "HMI-data".Bin4Breed, 1 s

HMI tags "Inputs"
   "Start_pos" : Bool = PLC Start_pos AT %I0.0, 1 s
   "Size_measure_pos" : Bool = PLC Size_measure_pos AT %I0.1, 1 s
   "Weight_mes_pos" : Bool = PLC Weight_mes_pos AT %I0.2, 1 s
   "Servo_table_pos" : Bool = PLC Servo_table_pos AT %I0.3, 1 s
   "Metal_sensor" : Bool = PLC Metal_sensor AT %I0.4, 1 s
   "Grip_cyl_end_ext" : Bool = PLC Grip_cyl_end_ext AT %I0.5, 1 s
   "Grip_cyl_end_ret" : Bool = PLC Grip_cyl_end_ret AT %I0.6, 1 s
   "Bin1_cyl_ext" : Bool = PLC Cyl_at_table_ext AT %I0.7, 1 s
   "Bin1_cyl_ret" : Bool = PLC Cyl_at_table_ret AT %I1.0, 1 s
   "ES1" : Bool = PLC ES1 AT %I1.7, 1 s
   "ES2" : Bool = PLC ES2 AT %I2.0, 1 s
   "Size_measure" : Int = PLC Size_measure AT %IW0, 1 s
   "Load_cell" : Int = PLC Load_cell AT %IW2, 1 s

HMI tags "Outputs"
   "Green_light" : Bool = PLC Green_light AT %Q4.0, 1 s
   "Yellow_light" : Bool = PLC Yellow_light AT %Q4.1, 1 s
   "Red_light" : Bool = PLC Red_light AT %Q4.2, 1 s
   "Move_grip_cyl_end_fwd" : Bool = PLC Move_grip_cyl_end_fwd AT %Q4.3, 1 s
   "Move_grip_cyl_end_bwd" : Bool = PLC Move_grip_cyl_end_bwd AT %Q4.4, 1 s
   "Conveyor_forward" : Bool = PLC Conveyor_forward AT %Q5.5, 1 s
   "Conveyor_backward" : Bool = PLC Conveyor_backward AT %Q5.6, 1 s
   "Move_cyl_at_table_fwd" : Bool = PLC Move_cyl_at_table_fwd AT %Q4.5, 1 s
   "Move_cyl_at_table_bwd" : Bool = PLC Move_cyl_at_table_bwd AT %Q4.6, 1 s
   "Move_grip_cyl_start_fwd(1)" : Bool = PLC Move_grip_cyl_start_fwd AT %Q5.7, 1 s
   "Move_grip_cyl_start_bwd" : Bool = PLC Move_grip_cyl_start_bwd AT %Q6.0, 1 s
   "Blue_light" : Bool = PLC Blue_light AT %Q4.7, 1 s

screen "Root screen" 800x443, template "Template_1"
   on GenerateScreen: SetTag("Tag_ScreenNumber", 1)
   Switch "Switch_1" at 24,41 size 147x49; CaptionText 'Switch'; TextOff 'Manual'; TextOn 'Automatic'
      ProcessValue <- "HMI-data_AutomaticMode"
   TextField "Text field_1" at 24,14 size 197x23; Text 'Automatic/Manual'
   Button "Button_1" at 196,49 size 134x55; TextOff 'Start conveyor'
      on Click: SetBit("HMI-data_StartConveyor")
   Button "Button_2" at 351,49 size 132x55; TextOff 'Stop conveyor'
   IOField "I/O field_1" at 27,188 size 96x32; FormatPattern s99.9
      ProcessValue <- "HMI-data_SizeInCm"
   TextField "Text field_2" at 150,157 size 68x23; Text 'Metal'
   TextField "Text field_3" at 49,160 size 55x23; Text 'Size'
   IOField "I/O field_2" at 232,188 size 96x32; FormatPattern s99.9
      ProcessValue <- "HMI-data_WeightInKg"
   TextField "Text field_4" at 247,159 size 81x23; Text 'Weight'
   Button "Button_3" at 644,320 size 153x32; TextOff 'Servo motion'
      on Release: ActivateScreen("Servo-motion-screen", 0)
   Circle "Circle_1" at 153,179 size 48x48
      Appearance <- "HMI-data_MetalMaterial"
   Circle "Circle_2" at 453,176 size 48x48
      Appearance <- "HMI-data_TableAtHome"
   Circle "Circle_3" at 515,176 size 48x48
      Appearance <- "HMI-data_TableAtBin1"
   Circle "Circle_4" at 579,176 size 48x48
      Appearance <- "HMI-data_TableAtBin2"
   Circle "Circle_5" at 697,176 size 48x48
      Appearance <- "HMI-data_TableAtBin4"
   Circle "Circle_6" at 638,176 size 48x48
      Appearance <- "HMI-data_TableAtBin3"
   TextField "Text field_5" at 453,148 size 62x23; Text 'Home'
   TextField "Text field_6" at 515,148 size 51x23; Text 'Bin1'
   TextField "Text field_7" at 579,148 size 51x23; Text 'Bin2'
   TextField "Text field_8" at 639,148 size 51x23; Text 'Bin3'
   TextField "Text field_9" at 697,148 size 51x23; Text 'Bin4'
   TextField "Text field_10" at 518,36 size 70x23; Text '24V OK'
      Visibility <- "HMI-data_ControlSupplyOK"
   TextField "Text field_11" at 604,29 size 123x61; Text 'Item in the system'
      Visibility <- "HMI-data_ItemInTheSystem"
   Button "Button_4" at 472,321 size 153x32; TextOff 'Manual motion'
      on Release: ActivateScreen("Manual-motion-screen", 0)
   Button "Button_5" at 365,321 size 96x32; TextOff 'Inputs'
      on Release: ActivateScreen("Inputs-screen", 0)
   TextField "Text field_12" at 353,159 size 70x23; Text 'Breed'
   TextField "Text field_13" at 357,188 size 45x23; Text 'Bin1'
      Visibility <- "HMI-data_Bin1Breed"
   TextField "Text field_14" at 357,188 size 45x23; Text 'Bin2'
      Visibility <- "HMI-data_Bin2Breed"
   TextField "Text field_15" at 357,188 size 45x23; Text 'Bin3'
      Visibility <- "HMI-data_Bin3Breed"
   TextField "Text field_16" at 357,188 size 45x23; Text 'Bin4'
      Visibility <- "HMI-data_Bin4Breed"

Template "Template_1" 800x443
   Button "Exit" at 720,360 size 78x58; TextOff 'Exit'; PictureOff "ExitRuntime_TP700_Comfort_TR"; PictureOn "ExitRuntime_TP700_Comfort_TR"
      on Release: StopRuntime(0)
   Button "Template_Button" at 640,360 size 78x58; TextOff 'Text'
   Button "Template_Button_1" at 560,360 size 78x58; TextOff 'Text'
   Button "Template_Button_2" at 480,360 size 78x58; TextOff 'Text'
   Button "Template_Button_3" at 400,360 size 78x58; TextOff 'Text'
   Button "Template_Button_4" at 321,360 size 78x58; TextOff 'Text'
   Button "Template_Button_5" at 241,360 size 78x58; TextOff 'Text'
   Button "Template_Button_6" at 161,360 size 78x58; TextOff 'Text'
   Button "Template_Button_7" at 81,360 size 78x58; TextOff 'Text'
   Button "Start screen" at 1,360 size 78x58; TextOff 'Start screen'; PictureOff "NavigateHome_TP700_Comfort_TR"; PictureOn "NavigateHome_TP700_Comfort_TR"
      on Release: ActivateScreen("Root screen", 0)

screen "Servo-motion-screen" 800x443
   Button "Button_1" at 7,31 size 96x32; TextOff 'Jog+'
   Button "Button_2" at 7,79 size 96x32; TextOff 'Jog-'
   Button "Button_3" at 7,127 size 96x32; TextOff 'Home'
   Button "Button_4" at 7,176 size 96x32; TextOff 'Bin1'
   Button "Button_5" at 7,223 size 96x32; TextOff 'Bin2'
   Button "Button_6" at 5,271 size 96x32; TextOff 'Bin3'
   Button "Button_7" at 5,319 size 96x32; TextOff 'Bin4'
   Button "Button_8" at 660,377 size 130x36; TextOff 'Main screen'
      on Release: ActivateScreen("Root screen", 0)
   TextField "Text field_1" at 28,1 size 68x23; Text 'Servo'
   TextField "Text field_2" at 348,16 size 194x23; Text 'Save new position'
   TextField "Text field_3" at 135,25 size 86x23; Text 'Position:'
   IOField "I/O field_1" at 229,22 size 96x32; FormatPattern 9999999
   Button "Button_9" at 373,48 size 96x32; TextOff 'Bin1'
   Button "Button_10" at 373,104 size 96x32; TextOff 'Bin2'
   Button "Button_11" at 373,159 size 96x32; TextOff 'Bin3'
   Button "Button_12" at 373,205 size 96x32; TextOff 'Bin4'

screen "Manual-motion-screen" 800x443
   TextField "Text field_1" at 52,5 size 89x23; Text 'Cylinders'
   Switch "Switch_1" at 63,79 size 117x40; CaptionText 'Switch'; TextOff 'OFF'; TextOn 'ON'
      ProcessValue <- "Move_grip_cyl_start_fwd(1)"
   TextField "Text field_2" at 5,47 size 148x23; Text 'Start position'
   TextField "Text field_3" at 5,87 size 57x23; Text 'FWD'
   Switch "Switch_2" at 63,125 size 117x40; TextOn 'ON'; CaptionText 'Switch'; TextOff 'OFF'
      ProcessValue <- "Move_grip_cyl_start_bwd"
   TextField "Text field_4" at 5,133 size 59x23; Text 'BWD'
   Switch "Switch_3" at 67,211 size 117x40; TextOn 'ON'; CaptionText 'Switch'; TextOff 'OFF'
      ProcessValue <- "Move_grip_cyl_end_fwd"
   TextField "Text field_5" at 14,179 size 135x23; Text 'End position'
   TextField "Text field_6" at 9,219 size 57x23; Text 'FWD'
   Switch "Switch_4" at 67,257 size 117x40; TextOn 'ON'; CaptionText 'Switch'; TextOff 'OFF'
      ProcessValue <- "Move_grip_cyl_end_bwd"
   TextField "Text field_7" at 9,265 size 59x23; Text 'BWD'
   Switch "Switch_5" at 74,343 size 117x40; TextOn 'ON'; CaptionText 'Switch'; TextOff 'OFF'
      ProcessValue <- "Move_cyl_at_table_fwd"
   TextField "Text field_8" at 19,311 size 74x23; Text 'Table'
   TextField "Text field_9" at 16,351 size 57x23; Text 'FWD'
   Switch "Switch_6" at 74,389 size 117x40; TextOn 'ON'; CaptionText 'Switch'; TextOff 'OFF'
      ProcessValue <- "Move_cyl_at_table_bwd"
   TextField "Text field_10" at 16,397 size 59x23; Text 'BWD'
   TextField "Text field_11" at 283,7 size 72x23; Text 'Lights'
   Switch "Switch_7" at 254,37 size 117x40; TextOn 'Blue on'; CaptionText 'Switch'; TextOff 'Blue off'
      ProcessValue <- "Blue_light"
   Switch "Switch_8" at 256,81 size 117x40; TextOn 'Green on'; CaptionText 'Switch'; TextOff 'Green off'
      ProcessValue <- "Green_light"
   Switch "Switch_9" at 257,125 size 117x40; TextOn 'Yellow on'; CaptionText 'Switch'; TextOff 'Yellow off'
      ProcessValue <- "Yellow_light"
   Switch "Switch_10" at 258,170 size 117x40; TextOn 'Red on'; CaptionText 'Switch'; TextOff 'Red off'
      ProcessValue <- "Red_light"
   TextField "Text field_12" at 453,7 size 101x23; Text 'Conveyor'
   Switch "Switch_11" at 437,45 size 117x40; TextOn 'Fwd on'; CaptionText 'Switch'; TextOff 'Fwd off'
      ProcessValue <- "Conveyor_forward"
   Switch "Switch_12" at 437,92 size 117x40; TextOn 'Bwd on'; CaptionText 'Switch'; TextOff 'Bwd off'
      ProcessValue <- "Conveyor_backward"
   Button "Button_1" at 636,388 size 127x32; TextOff 'Main Screen'
      on Release: ActivateScreen("Root screen", 0)

screen "Inputs-screen" 800x443
   TextField "Text field_1" at 9,14 size 196x23; Text 'Control 24V button'
   TextField "Text field_2" at 9,48 size 164x23; Text 'E-stop button 1'
   TextField "Text field_3" at 10,83 size 164x23; Text 'E-stop button 2'
   TextField "Text field_4" at 10,117 size 176x23; Text 'Starting position'
   TextField "Text field_5" at 12,152 size 186x118; Text 'Gripping cylinder at start position retracted'
   TextField "Text field_6" at 320,9 size 158x80; Text 'Metal measure position'
   TextField "Text field_12" at 13,348 size 145x80; Text 'Size measure position'
   TextField "Text field_13" at 13,248 size 186x99; Text 'Gripping cylinder at start position extended'
   Button "Button_1" at 605,377 size 128x32; TextOff 'Main Screen'
      on Release: ActivateScreen("Root screen", 0)
*)